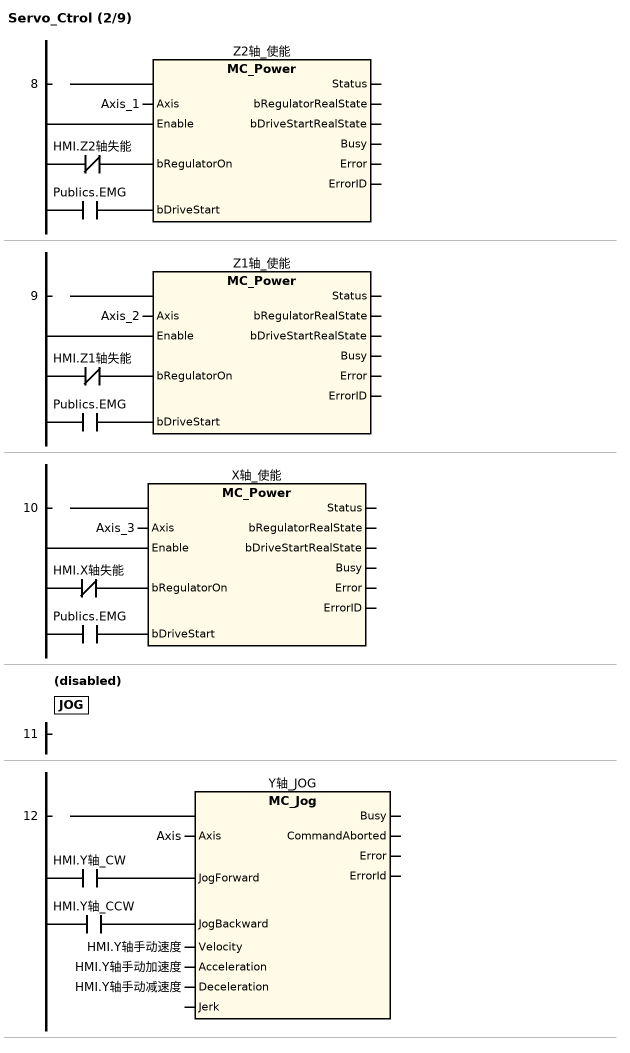
// NETWORK 8
Z2轴_使能(Axis := Axis_1, Enable := TRUE, bRegulatorOn := NOT HMI.Z2轴失能, bDriveStart := Publics.EMG); // MC_Power

// NETWORK 9
Z1轴_使能(Axis := Axis_2, Enable := TRUE, bRegulatorOn := NOT HMI.Z1轴失能, bDriveStart := Publics.EMG); // MC_Power

// NETWORK 10
X轴_使能(Axis := Axis_3, Enable := TRUE, bRegulatorOn := NOT HMI.X轴失能, bDriveStart := Publics.EMG); // MC_Power

// NETWORK 11 (disabled)
// label: JOG

// NETWORK 12
Y轴_JOG(
    Axis := Axis,
    JogForward := HMI.Y轴_CW,
    JogBackward := HMI.Y轴_CCW,
    Velocity := HMI.Y轴手动速度,
    Acceleration := HMI.Y轴手动加速度,
    Deceleration := HMI.Y轴手动减速度); // MC_Jog

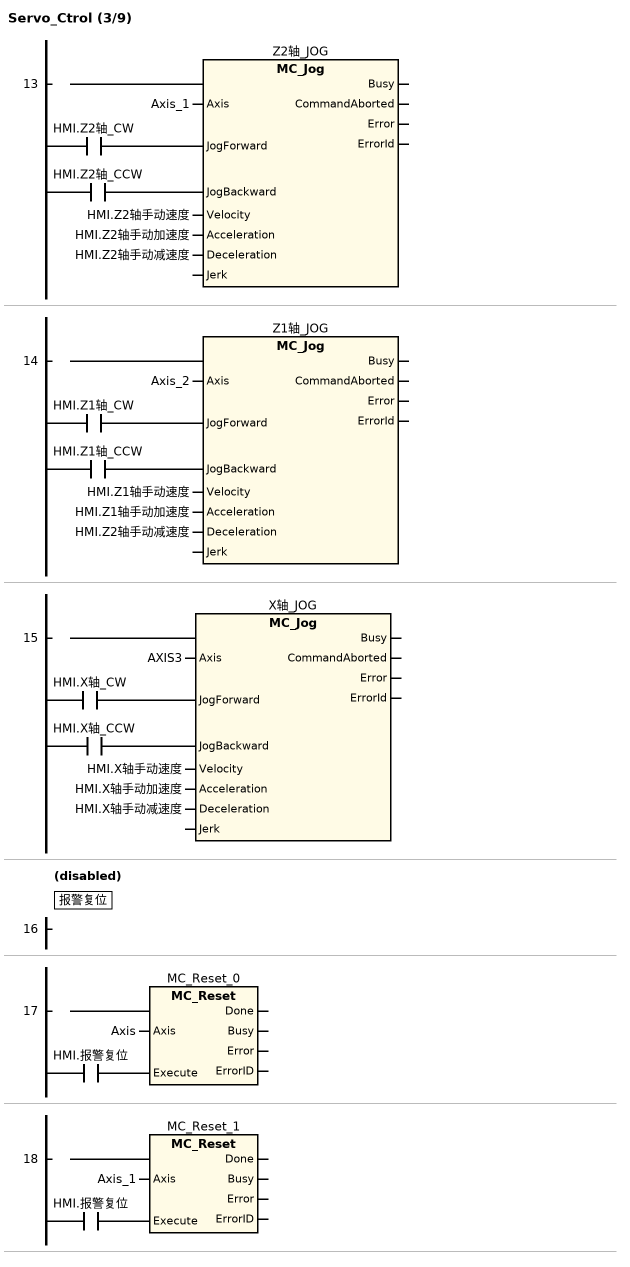
// NETWORK 13
Z2轴_JOG(
    Axis := Axis_1,
    JogForward := HMI.Z2轴_CW,
    JogBackward := HMI.Z2轴_CCW,
    Velocity := HMI.Z2轴手动速度,
    Acceleration := HMI.Z2轴手动加速度,
    Deceleration := HMI.Z2轴手动减速度); // MC_Jog

// NETWORK 14
Z1轴_JOG(
    Axis := Axis_2,
    JogForward := HMI.Z1轴_CW,
    JogBackward := HMI.Z1轴_CCW,
    Velocity := HMI.Z1轴手动速度,
    Acceleration := HMI.Z1轴手动加速度,
    Deceleration := HMI.Z2轴手动减速度); // MC_Jog

// NETWORK 15
X轴_JOG(
    Axis := AXIS3,
    JogForward := HMI.X轴_CW,
    JogBackward := HMI.X轴_CCW,
    Velocity := HMI.X轴手动速度,
    Acceleration := HMI.X轴手动加速度,
    Deceleration := HMI.X轴手动减速度); // MC_Jog

// NETWORK 16 (disabled)
// label: 报警复位

// NETWORK 17
MC_Reset_0(Axis := Axis, Execute := HMI.报警复位); // MC_Reset

// NETWORK 18
MC_Reset_1(Axis := Axis_1, Execute := HMI.报警复位); // MC_Reset

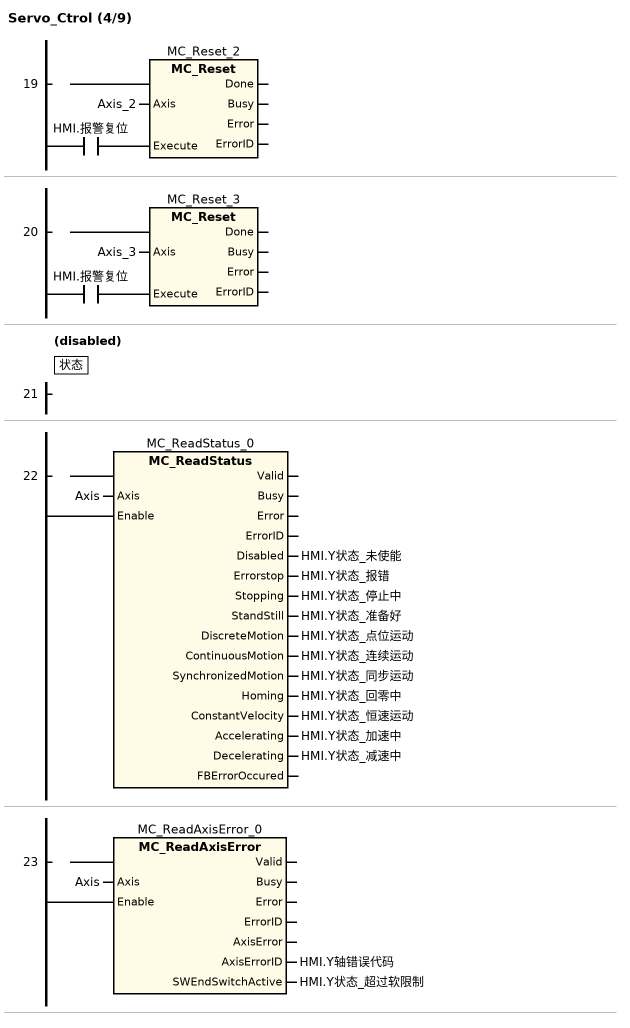
// NETWORK 19
MC_Reset_2(Axis := Axis_2, Execute := HMI.报警复位); // MC_Reset

// NETWORK 20
MC_Reset_3(Axis := Axis_3, Execute := HMI.报警复位); // MC_Reset

// NETWORK 21 (disabled)
// label: 状态

// NETWORK 22
MC_ReadStatus_0(
    Axis := Axis,
    Enable := TRUE,
    Disabled => HMI.Y状态_未使能,
    Errorstop => HMI.Y状态_报错,
    Stopping => HMI.Y状态_停止中,
    StandStill => HMI.Y状态_准备好,
    DiscreteMotion => HMI.Y状态_点位运动,
    ContinuousMotion => HMI.Y状态_连续运动,
    SynchronizedMotion => HMI.Y状态_同步运动,
    Homing => HMI.Y状态_回零中,
    ConstantVelocity => HMI.Y状态_恒速运动,
    Accelerating => HMI.Y状态_加速中,
    Decelerating => HMI.Y状态_减速中); // MC_ReadStatus

// NETWORK 23
MC_ReadAxisError_0(
    Axis := Axis,
    Enable := TRUE,
    AxisErrorID => HMI.Y轴错误代码,
    SWEndSwitchActive => HMI.Y状态_超过软限制); // MC_ReadAxisError

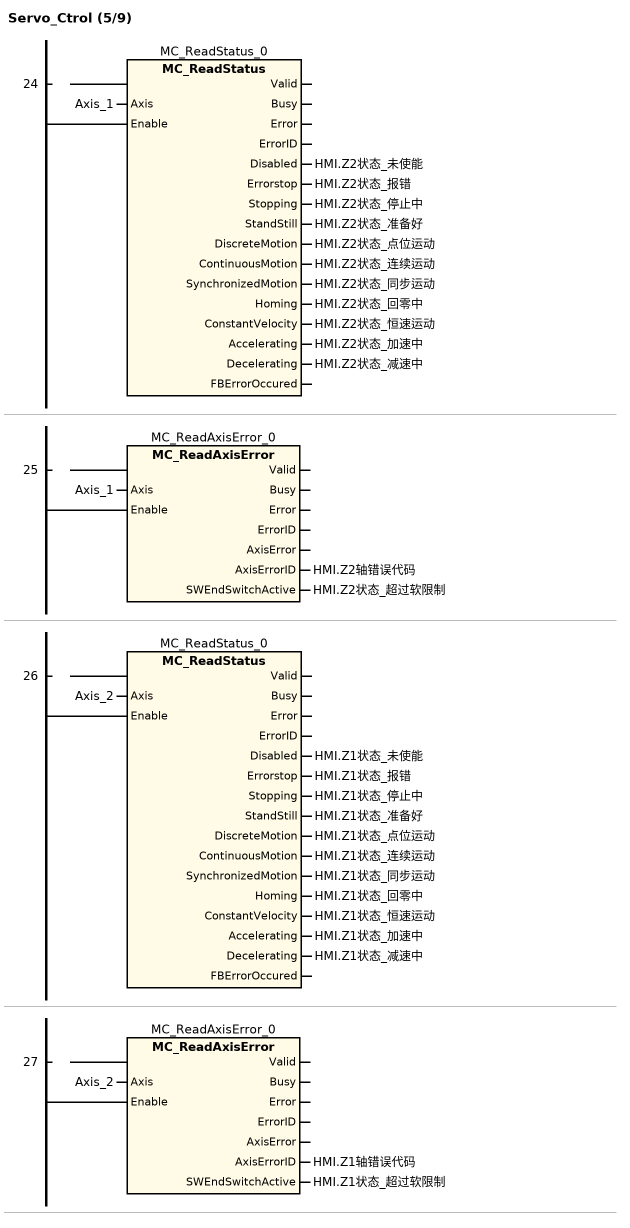
// NETWORK 24
MC_ReadStatus_0(
    Axis := Axis_1,
    Enable := TRUE,
    Disabled => HMI.Z2状态_未使能,
    Errorstop => HMI.Z2状态_报错,
    Stopping => HMI.Z2状态_停止中,
    StandStill => HMI.Z2状态_准备好,
    DiscreteMotion => HMI.Z2状态_点位运动,
    ContinuousMotion => HMI.Z2状态_连续运动,
    SynchronizedMotion => HMI.Z2状态_同步运动,
    Homing => HMI.Z2状态_回零中,
    ConstantVelocity => HMI.Z2状态_恒速运动,
    Accelerating => HMI.Z2状态_加速中,
    Decelerating => HMI.Z2状态_减速中); // MC_ReadStatus

// NETWORK 25
MC_ReadAxisError_0(
    Axis := Axis_1,
    Enable := TRUE,
    AxisErrorID => HMI.Z2轴错误代码,
    SWEndSwitchActive => HMI.Z2状态_超过软限制); // MC_ReadAxisError

// NETWORK 26
MC_ReadStatus_0(
    Axis := Axis_2,
    Enable := TRUE,
    Disabled => HMI.Z1状态_未使能,
    Errorstop => HMI.Z1状态_报错,
    Stopping => HMI.Z1状态_停止中,
    StandStill => HMI.Z1状态_准备好,
    DiscreteMotion => HMI.Z1状态_点位运动,
    ContinuousMotion => HMI.Z1状态_连续运动,
    SynchronizedMotion => HMI.Z1状态_同步运动,
    Homing => HMI.Z1状态_回零中,
    ConstantVelocity => HMI.Z1状态_恒速运动,
    Accelerating => HMI.Z1状态_加速中,
    Decelerating => HMI.Z1状态_减速中); // MC_ReadStatus

// NETWORK 27
MC_ReadAxisError_0(
    Axis := Axis_2,
    Enable := TRUE,
    AxisErrorID => HMI.Z1轴错误代码,
    SWEndSwitchActive => HMI.Z1状态_超过软限制); // MC_ReadAxisError

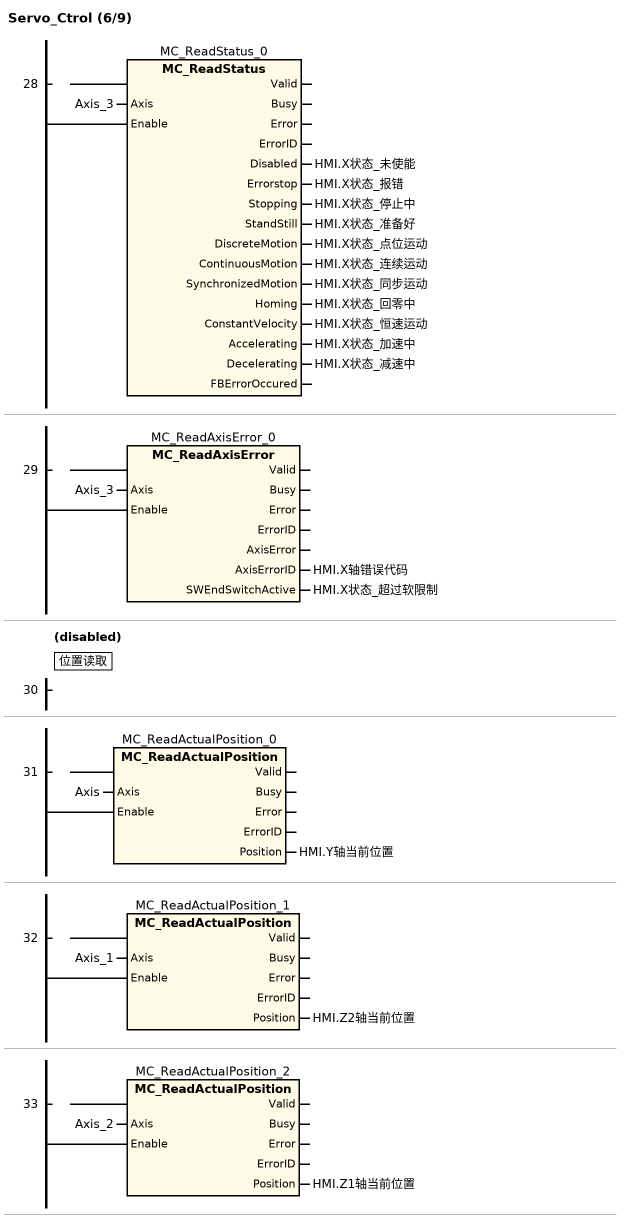
// NETWORK 28
MC_ReadStatus_0(
    Axis := Axis_3,
    Enable := TRUE,
    Disabled => HMI.X状态_未使能,
    Errorstop => HMI.X状态_报错,
    Stopping => HMI.X状态_停止中,
    StandStill => HMI.X状态_准备好,
    DiscreteMotion => HMI.X状态_点位运动,
    ContinuousMotion => HMI.X状态_连续运动,
    SynchronizedMotion => HMI.X状态_同步运动,
    Homing => HMI.X状态_回零中,
    ConstantVelocity => HMI.X状态_恒速运动,
    Accelerating => HMI.X状态_加速中,
    Decelerating => HMI.X状态_减速中); // MC_ReadStatus

// NETWORK 29
MC_ReadAxisError_0(
    Axis := Axis_3,
    Enable := TRUE,
    AxisErrorID => HMI.X轴错误代码,
    SWEndSwitchActive => HMI.X状态_超过软限制); // MC_ReadAxisError

// NETWORK 30 (disabled)
// label: 位置读取

// NETWORK 31
MC_ReadActualPosition_0(Axis := Axis, Enable := TRUE, Position => HMI.Y轴当前位置); // MC_ReadActualPosition

// NETWORK 32
MC_ReadActualPosition_1(Axis := Axis_1, Enable := TRUE, Position => HMI.Z2轴当前位置); // MC_ReadActualPosition

// NETWORK 33
MC_ReadActualPosition_2(Axis := Axis_2, Enable := TRUE, Position => HMI.Z1轴当前位置); // MC_ReadActualPosition

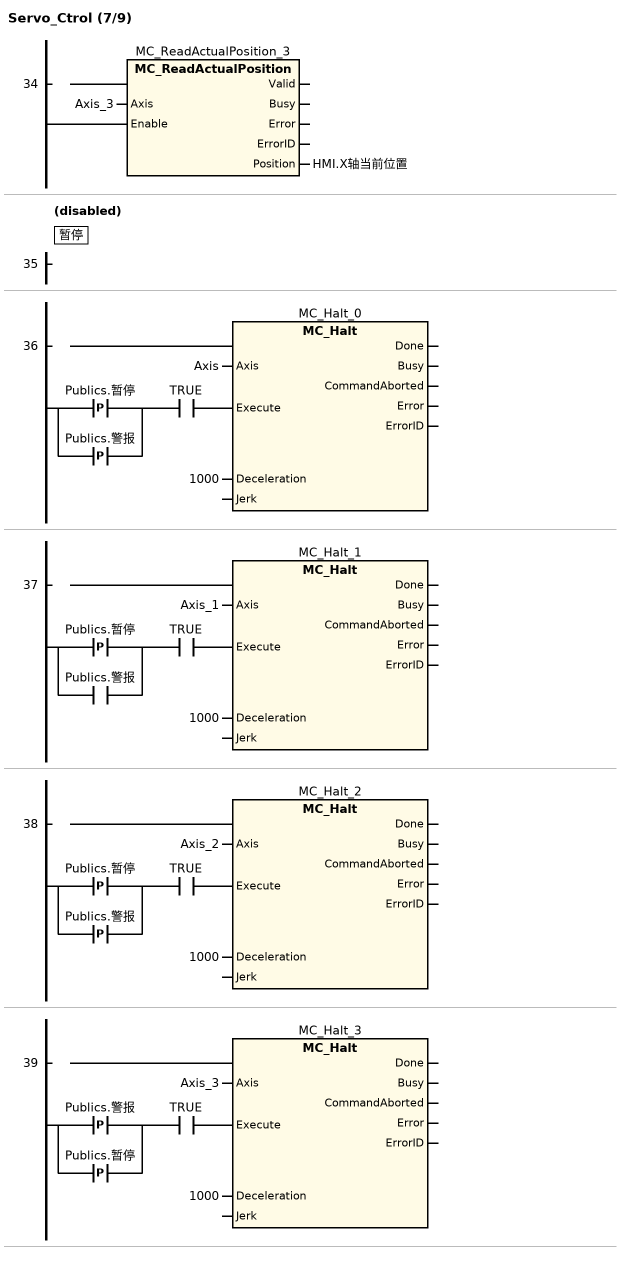
// NETWORK 34
MC_ReadActualPosition_3(Axis := Axis_3, Enable := TRUE, Position => HMI.X轴当前位置); // MC_ReadActualPosition

// NETWORK 35 (disabled)
// label: 暂停

// NETWORK 36
_rt1(CLK := Publics.暂停);
_rt2(CLK := Publics.警报);
MC_Halt_0(Axis := Axis, Execute := (_rt1.Q OR _rt2.Q) AND TRUE, Deceleration := 1000); // MC_Halt

// NETWORK 37
_rt3(CLK := Publics.暂停);
MC_Halt_1(Axis := Axis_1, Execute := (_rt3.Q OR Publics.警报) AND TRUE, Deceleration := 1000); // MC_Halt

// NETWORK 38
_rt4(CLK := Publics.暂停);
_rt5(CLK := Publics.警报);
MC_Halt_2(Axis := Axis_2, Execute := (_rt4.Q OR _rt5.Q) AND TRUE, Deceleration := 1000); // MC_Halt

// NETWORK 39
_rt6(CLK := Publics.警报);
_rt7(CLK := Publics.暂停);
MC_Halt_3(Axis := Axis_3, Execute := (_rt6.Q OR _rt7.Q) AND TRUE, Deceleration := 1000); // MC_Halt

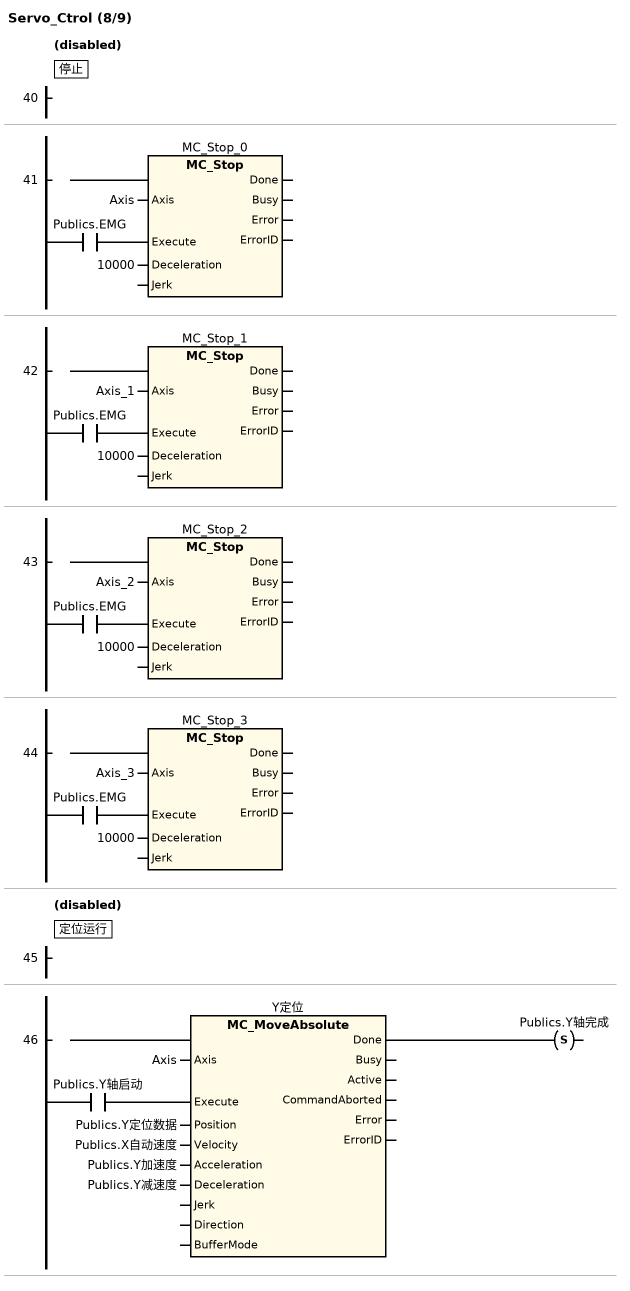
// NETWORK 40 (disabled)
// label: 停止

// NETWORK 41
MC_Stop_0(Axis := Axis, Execute := Publics.EMG, Deceleration := 10000); // MC_Stop

// NETWORK 42
MC_Stop_1(Axis := Axis_1, Execute := Publics.EMG, Deceleration := 10000); // MC_Stop

// NETWORK 43
MC_Stop_2(Axis := Axis_2, Execute := Publics.EMG, Deceleration := 10000); // MC_Stop

// NETWORK 44
MC_Stop_3(Axis := Axis_3, Execute := Publics.EMG, Deceleration := 10000); // MC_Stop

// NETWORK 45 (disabled)
// label: 定位运行

// NETWORK 46
Y定位(
    Axis := Axis,
    Execute := Publics.Y轴启动,
    Position := Publics.Y定位数据,
    Velocity := Publics.X自动速度,
    Acceleration := Publics.Y加速度,
    Deceleration := Publics.Y减速度); // MC_MoveAbsolute
Publics.Y轴完成 S= Y定位.Done;

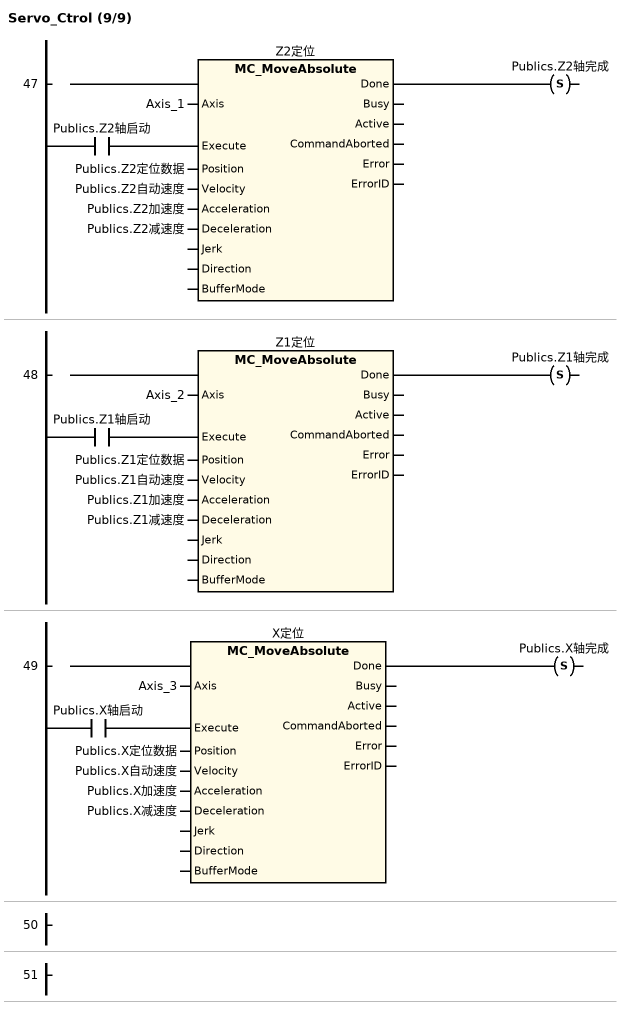
// NETWORK 47
Z2定位(
    Axis := Axis_1,
    Execute := Publics.Z2轴启动,
    Position := Publics.Z2定位数据,
    Velocity := Publics.Z2自动速度,
    Acceleration := Publics.Z2加速度,
    Deceleration := Publics.Z2减速度); // MC_MoveAbsolute
Publics.Z2轴完成 S= Z2定位.Done;

// NETWORK 48
Z1定位(
    Axis := Axis_2,
    Execute := Publics.Z1轴启动,
    Position := Publics.Z1定位数据,
    Velocity := Publics.Z1自动速度,
    Acceleration := Publics.Z1加速度,
    Deceleration := Publics.Z1减速度); // MC_MoveAbsolute
Publics.Z1轴完成 S= Z1定位.Done;

// NETWORK 49
X定位(
    Axis := Axis_3,
    Execute := Publics.X轴启动,
    Position := Publics.X定位数据,
    Velocity := Publics.X自动速度,
    Acceleration := Publics.X加速度,
    Deceleration := Publics.X减速度); // MC_MoveAbsolute
Publics.X轴完成 S= X定位.Done;

// NETWORK 50

// NETWORK 51

END_PROGRAM

// Device/Application/回原
PROGRAM 回原
VAR
	回原按钮: BOOL;
	回原条件: BOOL;
END_VAR

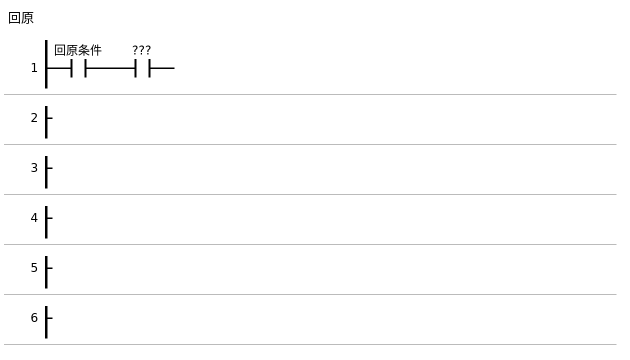
// NETWORK 1
(* 回原条件 AND ???; result not used *)

// NETWORK 2

// NETWORK 3

// NETWORK 4

// NETWORK 5

// NETWORK 6

END_PROGRAM

// Device/Application/ITF
INTERFACE ITF

END_INTERFACE

// Device/Application/FunctionBlock/FB_CylinderDouble
FUNCTION_BLOCK FB_CylinderDouble
VAR_IN_OUT
	///气缸控制、状态和报警
	stCylvar: CYLINDER_REF;
END_VAR
VAR_INPUT
	///安全条件
	xReady: BOOL;
	///报警复位
	xReset: BOOL;
	///手动控制,每on一次,则反转输出点状态
	xManuCmd: BOOL;
	///原位检测
	xBackSensor: BOOL;
	///到位检测
	xFrontSensor: BOOL;
	///手自动不一致报警无效
	xManuAlmDisable: BOOL;
	///原位检测无效
	xBackSensorDisable: BOOL;
	///到位检测无效	
	xFrontSensorDisable: BOOL;
	///原位延时	
	wBackDelay: WORD;
	///到位延时
	wFrontDelay: WORD;
END_VAR
VAR_OUTPUT
	///输出点,对应双控气缸原位电磁阀
	xOutputA: BOOL;
	///输出点,应双控气缸到位电磁阀
	xOutputB: BOOL;
	///未满足安全条件报警
	f_xNotRdyAlm: BOOL;
	///手自动不一致报警	
	f_xManuAlm: BOOL;
	///未在原位报警
	f_xBackAlm: BOOL;
	///未到位报警	
	f_xFrontAlm: BOOL;
	///气缸处于不受控制状态报警
	f_xUncontrolledAlm: BOOL;
END_VAR
VAR
	///获取自动控制的上升沿
	fbAutoRise: R_TRIG;
	///获取自动控制的下升沿
	fbAutoFall: F_TRIG;
	///获取手动控制的下升沿
	fbManuFall: F_TRIG;
	///获取复位信号的上升沿
	fbResetRise: R_TRIG;
	///原位状态延时,用于输出原位状态
	fbBackTon: TON;
	///到位状态延时,用于输出到位状态	
	fbFrontTon: TON;
	///获取原位状态下降沿
	fbBackFall: F_TRIG;
	///获取到位状态下降沿
	fbFrontFall: F_TRIG;
	///原位动作超时,用于输出未在原位位置报警
	fbBackWait: TON;
	///到位动作超时,用于输出未在原位位置报警
	fbFrontWait: TON;
END_VAR

   //初始化时返回原位
   IF  xReady AND stCylvar.xInit AND ( NOT xManuCmd ) THEN
	     xOutputA  := TRUE; 
         xOutputB  := FALSE;
		 f_xManuAlm  := FALSE;
		 stCylvar.xInit  := FALSE;	  	  	 	  
   END_IF	  
   
   //获取手动控制、自动控制的边沿信号
   fbManuFall(CLK:=xManuCmd , Q=> );
   fbAutoRise(CLK:=stCylvar.xAutoCmd , Q=> );
   fbAutoFall(CLK:=stCylvar.xAutoCmd , Q=> );
   
   //1,手动操作时，如果满足安全条件且未屏蔽手自动不一致报警时，则输出点A反转，输出点B取输出点A的反逻辑
   IF xReady AND (NOT xManuAlmDisable) AND fbManuFall.Q THEN
	   xOutputA  := NOT xOutputA; 
	   xOutputB  := NOT xOutputA;
	   
	//手动操作生效时，判断输出点状态与自动命令是否一致，不一致时,置位手动操作执行中报警；一致时复位该报警。
	//当因安全条件不满足导致自动命令未执行时，可通过手动操作控制其动作执行,此时手动操作并不引起手动操作执行中报警。
   	   IF (stCylvar.xAutoCmd AND (NOT xManuAlmDisable) ) XOR xOutputB THEN
   	   	    f_xManuAlm  :=TRUE;
   	   ELSE 
   	   	    f_xManuAlm  :=FALSE;
   	   END_IF
   END_IF
   //2,手动操作时，如果满足安全条件且屏蔽了手自动不一致报警时，则自动控制点反转、复位手自动不一致报警，  
    IF xReady AND  xManuAlmDisable AND fbManuFall.Q THEN
   	    stCylvar.xAutoCmd  := NOT stCylvar.xAutoCmd ;
		f_xManuAlm  :=FALSE;		  	 	
    END_IF
   
   //自动命令置位时，如满足安全条件，则输出点A复位、 输出点B置位。
   IF xReady AND fbAutoRise.Q THEN
   	    xOutputA  :=FALSE;
		xOutputB  :=TRUE;
		
   END_IF
   //自动命令复位时，如满足安全条件，则输出点A置位、 输出点B复位。
   IF xReady AND fbAutoFall.Q THEN
   	    xOutputA  :=TRUE;
		xOutputB  :=FALSE;		
   END_IF
   
   
   //到位状态输出
   fbFrontTon(IN:=( NOT xOutputA ) AND xOutputB AND ( xFrontSensor OR xFrontSensorDisable ) AND ( NOT xBackSensor ) , PT:= WORD_TO_TIME ( wFrontDelay *10 ), Q=> stCylvar.xIsFront, ET=> );
   
   //原位状态输出
   fbBackTon(IN:= xOutputA  AND ( NOT xOutputB) AND ( NOT xFrontSensor ) AND ( xBackSensor OR xBackSensorDisable ) , PT:= WORD_TO_TIME ( wBackDelay *10 ) , Q=> stCylvar.xIsBack, ET=> );
   
   
   //报警复位
   fbResetRise(CLK:= xReset, Q=> );
   IF fbResetRise.Q THEN
   	   f_xNotRdyAlm := FALSE;
	   f_xFrontAlm := FALSE;
	   f_xBackAlm := FALSE;
	   f_xUncontrolledAlm := FALSE;
   
   END_IF
   
   
   //未满足安全条件报警
   //当手动操作或自动命令状态发生改变时，如果不能满足安全条件，则输出未满足安全条件报警
   IF ( fbManuFall.Q OR fbAutoRise.Q OR fbAutoFall.Q ) AND ( NOT xReady ) THEN
   	   f_xNotRdyAlm := TRUE; 
   END_IF
   
   
   //未在原位报警
   //自动命令变OFF后(上电后气缸处于自由状态时不判断)，延时5秒，如果原位标志未变为ON、且未发生手动操作和安全条件报警，则输出未到原位报警
   fbBackWait(IN:= ( NOT stCylvar.xAutoCmd ) AND ( xOutputA OR xOutputB ) , PT:= T#5S , Q=> , ET=> );
   fbBackFall(CLK:= stCylvar.xIsBack , Q=> );
   IF (( fbBackWait.Q AND (NOT stCylvar.xIsBack )) OR (( NOT stCylvar.xAutoCmd ) AND fbBackFall.Q )) AND  ( NOT f_xManuAlm ) AND  ( NOT f_xNotRdyAlm ) THEN
   	    f_xBackAlm := TRUE;
   END_IF
   
   
   //未在到位报警
   //自动命令变ON后，延时5秒，如果到位标志未变为ON、且未发生手动操作和安全条件报警，则输出未到位报警
   fbFrontWait(IN:= stCylvar.xAutoCmd , PT:= T#5S , Q=> , ET=> );
   fbFrontFall(CLK:= stCylvar.xIsFront, Q=> );
   IF ( ( fbFrontWait.Q AND ( NOT stCylvar.xIsFront ) ) OR (stCylvar.xAutoCmd AND fbFrontFall.Q )) AND ( NOT f_xManuAlm ) AND ( NOT f_xNotRdyAlm ) THEN
   	    f_xFrontAlm := TRUE;   
   END_IF      
   
   
   //不受控状态报警
   IF NOT ( xOutputA OR xOutputB ) THEN
   	    f_xUncontrolledAlm := TRUE;
   END_IF

END_FUNCTION_BLOCK
